{attribute 'qualified_only'}
VAR_GLOBAL
END_VAR

(* stored: Version 1.1.0.1, ProductVersion 3.1.4024.4
   GVL Jog: Id {ebf25510-4b4a-4a3b-be8f-0a04e264c347} *)
